// TIA Portal V19 export
DATA_BLOCK "AO SCALING DB"   // DB6
{ S7_Optimized_Access := 'TRUE' }
// stored: MemoryReserve 100
   VAR
      SET : Struct
         "SYRUP MFG VESSEL SPEED" : Real;
         "PREMIXING VESSEL SPEED" : Real;
         "SUGAR VESSEL SPEED" : Real;
         SPARE : Real;
      END_STRUCT;
   END_VAR
   VAR RETAIN
      MIN : Struct
         "SYRUP MFG VESSEL SPEED" : Real;
         "PREMIXING VESSEL SPEED" : Real;
         "SUGAR VESSEL SPEED" : Real;
         SPARE : Real;
      END_STRUCT;
      MAX : Struct
         "SYRUP MFG VESSEL SPEED" : Real := 1450.0;
         "PREMIXING VESSEL SPEED" : Real := 1450.0;
         "SUGAR VESSEL SPEED" : Real := 1450.0;
         SPARE : Real;
      END_STRUCT;
   END_VAR
   VAR
      PV : Struct
         "SYRUP MFG VESSEL SPEED" : Real;
         "PREMIXING VESSEL SPEED" : Real;
         "SUGAR VESSEL SPEED" : Real;
         SPARE : Real;
      END_STRUCT;
   END_VAR
BEGIN
END_DATA_BLOCK
